FUNCTION_BLOCK FB_SendDataQue
VAR

END_VAR
VAR (*DATA ACCESS BY SERVAL TASK*)
	bSendQueFill		: BOOL;
	bSendQueLock		: BOOL;
	SendQue				: ARRAY[1..GVL.MaxDataLen] OF BYTE;
	
	GetDataFailCNT		: UDINT := 0;
	PutDataFailCNT		: UDINT := 0;
END_VAR

VAR_OUTPUT
	bGetData			: BOOL;
END_VAR

METHOD GetFromQue : BOOL
VAR_INPUT
	DataBuff 		: POINTER TO ARRAY[1..GVL.MaxDataLen] OF BYTE;
END_VAR
IF TestAndSet(bSendQueLock)THEN
	IF bSendQueFill THEN
		memcpy(DataBuff,ADR(SendQue),GVL.MaxDataLen);	
		bSendQueFill:= FALSE;
		bGetData := TRUE;
		GetDataFailCNT := 0;
	ELSE 
		memcpy(DataBuff,0,SIZEOF(DataBuff));
		GetDataFailCNT := GetDataFailCNT+1;
		bGetData := FALSE;
	END_IF
	bSendQueLock:= FALSE;	
ELSE
	//the que is emty, set buffer 0.
	memset(DataBuff,0,SIZEOF(DataBuff));
	GetDataFailCNT := GetDataFailCNT+1;
	bGetData := FALSE;
END_IF
END_METHOD

METHOD PutToQue : BOOL
VAR_INPUT
	DataBuff 		: POINTER TO ARRAY[1..GVL.MaxDataLen] OF BYTE;
END_VAR
IF TestAndSet(bSendQueLock) THEN
	memcpy(ADR(SendQue),DataBuff,GVL.MaxDataLen);
	bSendQueFill:= TRUE;
	PutDataFailCNT := 0;
	
	bSendQueLock:= FALSE;
ELSE
	PutDataFailCNT := PutDataFailCNT + 1;
END_IF
END_METHOD

METHOD Reset : BOOL
VAR_INPUT
END_VAR
IF TestAndSet(bSendQueLock) THEN
	bSendQueFill:= FALSE;
	bGetData := FALSE;
	
	bSendQueLock:= FALSE;	
END_IF
END_METHOD

END_FUNCTION_BLOCK

(* stored: Version 1.1.0.1, ProductVersion 3.1.4022.12
   POU FB_SendDataQue: Id {9e23bc2c-a2c1-4a8c-ae27-e57744d509a3}, SpecialFunc None
   Method GetFromQue: Id {32989078-c026-44fb-a2d9-c267dd20c336}
   Method PutToQue: Id {256b9177-5167-48da-a7fa-62dc46dd6936}
   Method Reset: Id {fe90a66d-742a-498f-a873-e8176e784b55} *)
